FUNCTION_BLOCK E_T_FF_SR_SYM_INIT (* Event-driven bistable and Toggle, symmetric Start-Up Behaviour and INIT *)
  (* Standard: 61499-1 Annex A; Description: Copyright (c) 2017 fortiss GmbH, HR Agrartechnik GmbH This program and the accompanying materials are made available under the terms of the Eclipse Public License 2.0 which is available at https://www.eclipse.org/legal/epl-2.0/ SPDX-License-Identifier: EPL-2.0 *)
  (* Version 1.0, 2026-05-12, Franz Höpfinger, HR Agrartechnik GmbH, initial API and implementation and/or initial documentation *)
  PACKAGE iec61499::events;
  IMPORT eclipse4diac::core::TypeHash;
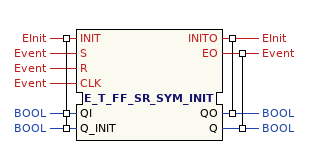
  EVENT_INPUT
    INIT : EInit WITH QI, Q_INIT; (* Initialization Request *)
    S; (* Set output Q *)
    R; (* Reset output Q *)
    CLK; (* Clock for triggering a output toggle *)
  END_EVENT
  EVENT_OUTPUT
    INITO : EInit WITH QO; (* Initialization Confirm *)
    EO WITH Q; (* Output Q has changed *)
  END_EVENT
  VAR_INPUT
    QI : BOOL; (* Input event qualifier *)
    Q_INIT : BOOL; (* Value of Q at INIT *)
  END_VAR
  VAR_OUTPUT
    QO : BOOL; (* Output event qualifier *)
    Q : BOOL; (* value of flip flop *)
  END_VAR
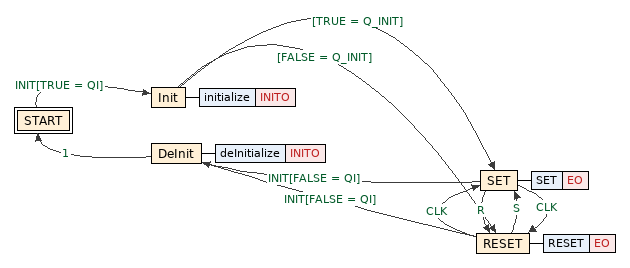
  EC_STATES
    START; (* Initial State *)
    Init : initialize -> INITO; (* Initialization *)
    DeInit : deInitialize -> INITO;
    SET : SET -> EO;
    RESET : RESET -> EO;
  END_STATES
  EC_TRANSITIONS
    SET TO RESET := R;
    RESET TO SET := S;
    SET TO RESET := CLK;
    RESET TO SET := CLK;
    START TO Init := INIT[TRUE = QI];
    Init TO RESET := [FALSE = Q_INIT];
    DeInit TO START := 1;
    RESET TO DeInit := INIT[FALSE = QI];
    SET TO DeInit := INIT[FALSE = QI];
    Init TO SET := [TRUE = Q_INIT];
  END_TRANSITIONS
  ALGORITHM initialize IN ST: (* Initialization algorithm *)
QO := QI;
  END_ALGORITHM
  ALGORITHM deInitialize IN ST: (* Normally executed algorithm *)
QO := FALSE;
  END_ALGORITHM
  ALGORITHM SET IN ST: (* SET algorithm *)
QO := QI;
IF TRUE = QI THEN
	(* only perform normal operation of QI is true *)
	Q := TRUE;
END_IF;
  END_ALGORITHM
  ALGORITHM RESET IN ST: (* RESET algorithm *)
QO := QI;
IF TRUE = QI THEN
	(* only perform normal operation of QI is true *)
	Q := FALSE;
END_IF;
  END_ALGORITHM
END_FUNCTION_BLOCK
